{attribute 'qualified_only'}
{attribute 'strict'}
TYPE E_BorderDashType :
(
	Solid := 0,
	RoundDot,
	SquareDot,
	Dash,
	LongDashDot
);
END_TYPE

(* stored: Version 1.1.0.1, ProductVersion 3.1.4024.12
   DUT E_BorderDashType: Id {52d7deba-4850-4e05-a3d3-e6836065ade5} *)
